// TIA Portal V21 export
FUNCTION_BLOCK "GestWatchdog_Incrementale"   // FB3, LAD
{ S7_Optimized_Access := 'TRUE' }
// stored: MemoryReserve 100, SetENOAutomatically false
   VAR_INPUT
      Watchdog_Recive : DInt;
      Reset : Bool;
   END_VAR
   VAR_OUTPUT
      Watchdog_Send : DInt;
   END_VAR
   VAR_IN_OUT
      Allarme : Bool;
   END_VAR
   VAR
      Watchdog_Prec : DInt;
      TimerAllarme : "Std_stTimer";
   END_VAR
BEGIN

REGION Network 1 (SCL)
   IF #Watchdog_Recive > 1000000 THEN
       #Watchdog_Send += 1;
       IF #Watchdog_Send > 1000000 THEN
           #Watchdog_Send := 0;
       END_IF;
   ELSE
       #Watchdog_Send := #Watchdog_Recive + 1;
   END_IF;

   #TimerAllarme.Preset := 6.0;
END_REGION

REGION Network 2: Allarme di comunicazione
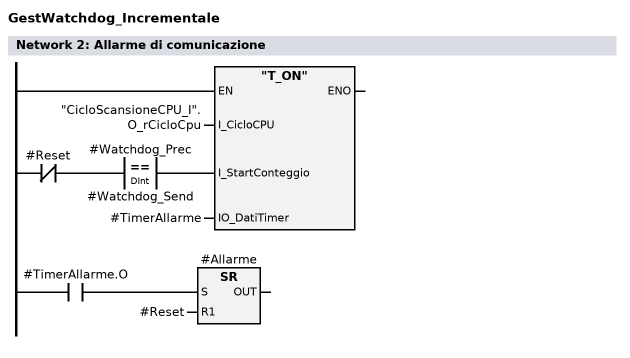
   RUNG wire#powerrail
      "T_ON"(I_StartConteggio := wire#w1, I_CicloCPU := "CicloScansioneCPU_I".O_rCicloCpu, IO_DatiTimer := #TimerAllarme)
   END_RUNG
   RUNG wire#powerrail
      I_Contact( #Reset )
      { S7_Templates := "SrcType := DInt" } EQ_Contact(in1 := #Watchdog_Prec, in2 := #Watchdog_Send)
   END_RUNG wire#w1
   RUNG wire#powerrail
      Contact( #TimerAllarme.O )
      S_SR(operand := #Allarme, r1 := #Reset)
   END_RUNG
   // the same network as SCL:
   "T_ON"(I_CicloCPU := "CicloScansioneCPU_I".O_rCicloCpu,
          I_StartConteggio := NOT #Reset AND (#Watchdog_Prec = #Watchdog_Send),
          IO_DatiTimer := #TimerAllarme);
   IF #TimerAllarme.O THEN
       #Allarme := TRUE;   // SR flip-flop
   END_IF;
   IF #Reset THEN #Allarme := FALSE; END_IF;
END_REGION

REGION Network 3 (SCL)
   #Watchdog_Prec := #Watchdog_Send;
END_REGION
END_FUNCTION_BLOCK
